FUNCTION_BLOCK PositionToDegree
VAR_INPUT
	MaxPosition : LREAL;
	MaxSteeringAngle : INT;
	Position : LREAL;
END_VAR
VAR_OUTPUT
	Deg : LREAL;
END_VAR
VAR
END_VAR

IF (Position > 0 OR Position < 0) THEN
	Deg := (MaxSteeringAngle/MaxPosition)*Position;
ELSIF (Position = 0) THEN
	Deg := 0;		
END_IF

END_FUNCTION_BLOCK

(* stored: Version 1.1.0.1, ProductVersion 3.1.4024.3
   POU PositionToDegree: Id {254cc25f-d883-4ebb-aede-8f10272b5caa}, SpecialFunc None *)
